// TIA Portal project "motors8" (V17)

(* hardware
DEVICE "S7-1500/ET200MP station_1"  S7-1500 station
   slot 0: "Rail_0"  Rack  6ES7 590-1***0-0AA0
   slot 1: "PLC_1"  CPU 1515-2 PN  6ES7 515-2AM02-0AB0  V2.9
      slot 3: "CPU display_1"  6ES7591-1BA00-0AA0
      slot 32768: "PROFINET interface_1"  X1
         slot 32769: "Port_1"  X1 P1
         slot 32770: "Port_2"  X1 P2
      slot 33024: "PROFINET interface_2"  X2
         slot 33025: "Port_1"  X2 P1
      slot 34817: "Virtual CP interface port_1"  Virtual CP interface port  Virtual CP interface port
   slot 2: "DQ 32x24VDC/0.5A BA_1"  DQ 32x24VDC/0.5A BA  6ES7 522-1BL10-0AA0  V1.1
DEVICE "PC-System_1"  SIMATIC PC station
   slot 0: "SIMATIC PC station"  Rail  SIMATIC PC-Station  V1.0
      slot 125: "Stationmanager"  Station_Manager  V6.0.4
   slot 1: "HMI_RT_1"  WinCC RT Advanced  6AV2 104-0xxxx-xxxx  17.0.0.0
      slot 33792: "Computer interface"  Host interface
   slot 2: "IE general_1"  IE General  IE_CP  V8.2.0
      slot 1: "PROFINET interface"  IEGeneral.Interface.8.2.0
*)

// ===== PLC "PLC_1"  CPU 1515-2 PN =====

VAR_GLOBAL   // PLC tag table "Default tag table"
   "MOTOR1" AT %Q0.0 : Bool;
   "MOTOR2" AT %Q0.1 : Bool;
   "MOTOR3" AT %Q0.2 : Bool;
   "MOTOR4" AT %Q0.3 : Bool;
   "MOTOR5" AT %Q0.4 : Bool;
   "MOTOR6" AT %Q0.5 : Bool;
   "MOTOR7" AT %Q0.6 : Bool;
   "MOTOR8" AT %Q0.7 : Bool;
END_VAR

TYPE "MotorLibrary"
   STRUCT
      "BREAKER ON" : Bool;
      OVERLOAD : Bool;
      CONTACTOR : Bool;
      "LED RUN" : Bool;
      "LED STOP" : Bool;
      "LED OVERLOAD" : Bool;
      "EMERGENCY STOP" : Bool;
      "START BUTTON" : Bool;
      "STOP BUTTON" : Bool;
      "RESET OVERLOAD" : Bool;
   END_STRUCT;
END_TYPE

DATA_BLOCK "MOTORsDB"   // DB1
{ S7_Optimized_Access := 'FALSE' }
VERSION : 0.1
   VAR
      M1 : "MotorLibrary";
      M2 : "MotorLibrary";
      M3 : "MotorLibrary";
      M4 : "MotorLibrary";
      M5 : "MotorLibrary";
      M6 : "MotorLibrary";
      M7 : "MotorLibrary";
      M8 : "MotorLibrary";
   END_VAR
BEGIN
END_DATA_BLOCK

DATA_BLOCK "FB_MOTOR1"   // DB2
{ S7_Optimized_Access := 'TRUE' }
VERSION : 0.1
// stored: InstanceOfName MOTORsLOGIC
"MOTORsLOGIC"
BEGIN
END_DATA_BLOCK

DATA_BLOCK "FB_MOTOR2"   // DB3
{ S7_Optimized_Access := 'TRUE' }
VERSION : 0.1
// stored: InstanceOfName MOTORsLOGIC
"MOTORsLOGIC"
BEGIN
END_DATA_BLOCK

DATA_BLOCK "FB_MOTOR3"   // DB4
{ S7_Optimized_Access := 'TRUE' }
VERSION : 0.1
// stored: InstanceOfName MOTORsLOGIC
"MOTORsLOGIC"
BEGIN
END_DATA_BLOCK

DATA_BLOCK "FB_MOTOR4"   // DB5
{ S7_Optimized_Access := 'TRUE' }
VERSION : 0.1
// stored: InstanceOfName MOTORsLOGIC
"MOTORsLOGIC"
BEGIN
END_DATA_BLOCK

DATA_BLOCK "FB_MOTOR5"   // DB6
{ S7_Optimized_Access := 'TRUE' }
VERSION : 0.1
// stored: InstanceOfName MOTORsLOGIC
"MOTORsLOGIC"
BEGIN
END_DATA_BLOCK

DATA_BLOCK "FB_MOTOR6"   // DB7
{ S7_Optimized_Access := 'TRUE' }
VERSION : 0.1
// stored: InstanceOfName MOTORsLOGIC
"MOTORsLOGIC"
BEGIN
END_DATA_BLOCK

DATA_BLOCK "FB_MOTOR7"   // DB8
{ S7_Optimized_Access := 'TRUE' }
VERSION : 0.1
// stored: InstanceOfName MOTORsLOGIC
"MOTORsLOGIC"
BEGIN
END_DATA_BLOCK

DATA_BLOCK "FB_MOTOR8"   // DB9
{ S7_Optimized_Access := 'TRUE' }
VERSION : 0.1
// stored: InstanceOfName MOTORsLOGIC
"MOTORsLOGIC"
BEGIN
END_DATA_BLOCK

FUNCTION_BLOCK "MOTORsLOGIC"   // FB1, LAD
{ S7_Optimized_Access := 'TRUE' }
VERSION : 0.1
   VAR_INPUT
      "BREAKER ON" : Bool;
      "EMERGENCY STOP" : Bool;
      "START BUTTON" : Bool;
      "STOP BUTTON" : Bool;
      "OVERLOAD RELAY" : Bool;
      "RESET OVERLOAD" : Bool;
   END_VAR
   VAR_OUTPUT
      CONTACTOR : Bool;
      "PLC OUTPUT" : Bool;
      "LED STOP" : Bool;
      "LED RUN" : Bool;
      "LED OVERLOAD" : Bool;
   END_VAR
   VAR_TEMP   // added for the SCL form of the ladder/FBD networks
      _w1 : Bool;
   END_VAR
BEGIN

REGION Network 1: Motors Logic Control
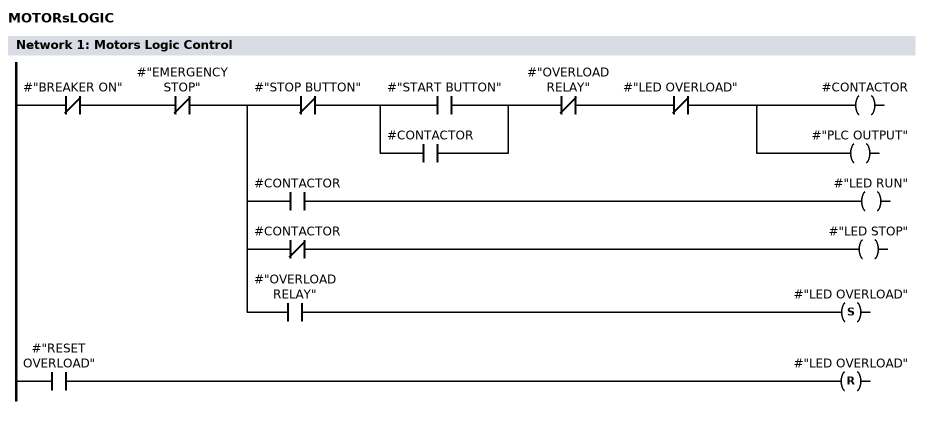
   RUNG wire#powerrail
      I_Contact( #"BREAKER ON" )
      I_Contact( #"EMERGENCY STOP" )
      wire#w1
      I_Contact( #"STOP BUTTON" )
      wire#w2
      Contact( #"START BUTTON" )
      wire#w3
      I_Contact( #"OVERLOAD RELAY" )
      I_Contact( #"LED OVERLOAD" )
      wire#w4
      Coil( #CONTACTOR )
   END_RUNG
   RUNG wire#w2
      Contact( #CONTACTOR )
   END_RUNG wire#w3
   RUNG wire#w4
      Coil( #"PLC OUTPUT" )
   END_RUNG
   RUNG wire#w1
      Contact( #CONTACTOR )
      Coil( #"LED RUN" )
   END_RUNG
   RUNG wire#w1
      I_Contact( #CONTACTOR )
      Coil( #"LED STOP" )
   END_RUNG
   RUNG wire#w1
      Contact( #"OVERLOAD RELAY" )
      S_Coil( #"LED OVERLOAD" )
   END_RUNG
   RUNG wire#powerrail
      Contact( #"RESET OVERLOAD" )
      R_Coil( #"LED OVERLOAD" )
   END_RUNG
   // the same network as SCL:
   #_w1 := NOT #"BREAKER ON" AND NOT #"EMERGENCY STOP";
   #CONTACTOR := #_w1 AND NOT #"STOP BUTTON" AND (#"START BUTTON" OR #CONTACTOR) AND NOT #"OVERLOAD RELAY" AND NOT #"LED OVERLOAD";
   #"PLC OUTPUT" := #CONTACTOR;
   #"LED RUN" := #_w1 AND #CONTACTOR;
   #"LED STOP" := #_w1 AND NOT #CONTACTOR;
   IF #_w1 AND #"OVERLOAD RELAY" THEN #"LED OVERLOAD" := TRUE; END_IF;
   IF #"RESET OVERLOAD" THEN #"LED OVERLOAD" := FALSE; END_IF;
END_REGION
END_FUNCTION_BLOCK

ORGANIZATION_BLOCK "Main"   // OB1, LAD, ProgramCycle
TITLE = "Main Program Sweep (Cycle)"
{ S7_Optimized_Access := 'TRUE' }
VERSION : 0.1
   VAR_INPUT
      Initial_Call : Bool;   // Initial call of this OB
      Remanence : Bool;   // =True, if remanent data are available
   END_VAR
BEGIN

REGION Network 1: MOTOR1
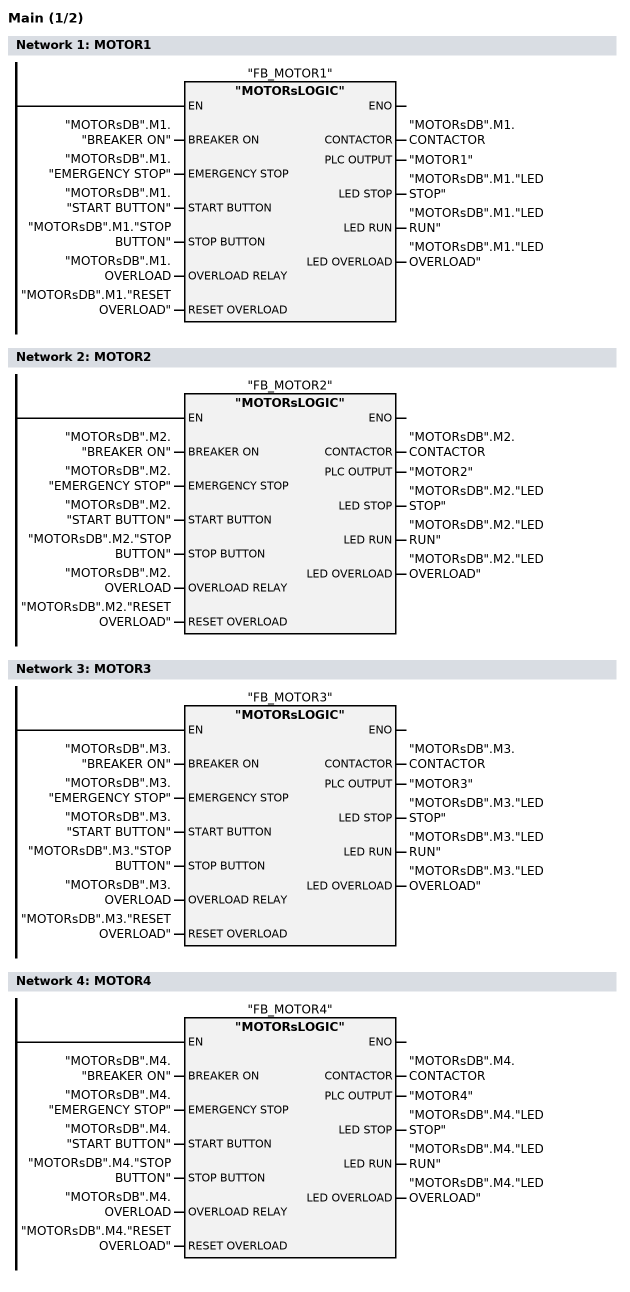
   RUNG wire#powerrail
      "FB_MOTOR1"("BREAKER ON" := "MOTORsDB".M1."BREAKER ON", "EMERGENCY STOP" := "MOTORsDB".M1."EMERGENCY STOP", "START BUTTON" := "MOTORsDB".M1."START BUTTON", "STOP BUTTON" := "MOTORsDB".M1."STOP BUTTON", "OVERLOAD RELAY" := "MOTORsDB".M1.OVERLOAD, "RESET OVERLOAD" := "MOTORsDB".M1."RESET OVERLOAD", CONTACTOR => "MOTORsDB".M1.CONTACTOR, "PLC OUTPUT" => "MOTOR1", "LED STOP" => "MOTORsDB".M1."LED STOP", "LED RUN" => "MOTORsDB".M1."LED RUN", "LED OVERLOAD" => "MOTORsDB".M1."LED OVERLOAD")
   END_RUNG
   // the same network as SCL:
   "FB_MOTOR1"("BREAKER ON" := "MOTORsDB".M1."BREAKER ON",   // "MOTORsLOGIC"
               "EMERGENCY STOP" := "MOTORsDB".M1."EMERGENCY STOP",
               "START BUTTON" := "MOTORsDB".M1."START BUTTON",
               "STOP BUTTON" := "MOTORsDB".M1."STOP BUTTON",
               "OVERLOAD RELAY" := "MOTORsDB".M1.OVERLOAD,
               "RESET OVERLOAD" := "MOTORsDB".M1."RESET OVERLOAD",
               CONTACTOR => "MOTORsDB".M1.CONTACTOR,
               "PLC OUTPUT" => "MOTOR1",
               "LED STOP" => "MOTORsDB".M1."LED STOP",
               "LED RUN" => "MOTORsDB".M1."LED RUN",
               "LED OVERLOAD" => "MOTORsDB".M1."LED OVERLOAD");
END_REGION

REGION Network 2: MOTOR2
   RUNG wire#powerrail
      "FB_MOTOR2"("BREAKER ON" := "MOTORsDB".M2."BREAKER ON", "EMERGENCY STOP" := "MOTORsDB".M2."EMERGENCY STOP", "START BUTTON" := "MOTORsDB".M2."START BUTTON", "STOP BUTTON" := "MOTORsDB".M2."STOP BUTTON", "OVERLOAD RELAY" := "MOTORsDB".M2.OVERLOAD, "RESET OVERLOAD" := "MOTORsDB".M2."RESET OVERLOAD", CONTACTOR => "MOTORsDB".M2.CONTACTOR, "PLC OUTPUT" => "MOTOR2", "LED STOP" => "MOTORsDB".M2."LED STOP", "LED RUN" => "MOTORsDB".M2."LED RUN", "LED OVERLOAD" => "MOTORsDB".M2."LED OVERLOAD")
   END_RUNG
   // the same network as SCL:
   "FB_MOTOR2"("BREAKER ON" := "MOTORsDB".M2."BREAKER ON",   // "MOTORsLOGIC"
               "EMERGENCY STOP" := "MOTORsDB".M2."EMERGENCY STOP",
               "START BUTTON" := "MOTORsDB".M2."START BUTTON",
               "STOP BUTTON" := "MOTORsDB".M2."STOP BUTTON",
               "OVERLOAD RELAY" := "MOTORsDB".M2.OVERLOAD,
               "RESET OVERLOAD" := "MOTORsDB".M2."RESET OVERLOAD",
               CONTACTOR => "MOTORsDB".M2.CONTACTOR,
               "PLC OUTPUT" => "MOTOR2",
               "LED STOP" => "MOTORsDB".M2."LED STOP",
               "LED RUN" => "MOTORsDB".M2."LED RUN",
               "LED OVERLOAD" => "MOTORsDB".M2."LED OVERLOAD");
END_REGION

REGION Network 3: MOTOR3
   RUNG wire#powerrail
      "FB_MOTOR3"("BREAKER ON" := "MOTORsDB".M3."BREAKER ON", "EMERGENCY STOP" := "MOTORsDB".M3."EMERGENCY STOP", "START BUTTON" := "MOTORsDB".M3."START BUTTON", "STOP BUTTON" := "MOTORsDB".M3."STOP BUTTON", "OVERLOAD RELAY" := "MOTORsDB".M3.OVERLOAD, "RESET OVERLOAD" := "MOTORsDB".M3."RESET OVERLOAD", CONTACTOR => "MOTORsDB".M3.CONTACTOR, "PLC OUTPUT" => "MOTOR3", "LED STOP" => "MOTORsDB".M3."LED STOP", "LED RUN" => "MOTORsDB".M3."LED RUN", "LED OVERLOAD" => "MOTORsDB".M3."LED OVERLOAD")
   END_RUNG
   // the same network as SCL:
   "FB_MOTOR3"("BREAKER ON" := "MOTORsDB".M3."BREAKER ON",   // "MOTORsLOGIC"
               "EMERGENCY STOP" := "MOTORsDB".M3."EMERGENCY STOP",
               "START BUTTON" := "MOTORsDB".M3."START BUTTON",
               "STOP BUTTON" := "MOTORsDB".M3."STOP BUTTON",
               "OVERLOAD RELAY" := "MOTORsDB".M3.OVERLOAD,
               "RESET OVERLOAD" := "MOTORsDB".M3."RESET OVERLOAD",
               CONTACTOR => "MOTORsDB".M3.CONTACTOR,
               "PLC OUTPUT" => "MOTOR3",
               "LED STOP" => "MOTORsDB".M3."LED STOP",
               "LED RUN" => "MOTORsDB".M3."LED RUN",
               "LED OVERLOAD" => "MOTORsDB".M3."LED OVERLOAD");
END_REGION

REGION Network 4: MOTOR4
   RUNG wire#powerrail
      "FB_MOTOR4"("BREAKER ON" := "MOTORsDB".M4."BREAKER ON", "EMERGENCY STOP" := "MOTORsDB".M4."EMERGENCY STOP", "START BUTTON" := "MOTORsDB".M4."START BUTTON", "STOP BUTTON" := "MOTORsDB".M4."STOP BUTTON", "OVERLOAD RELAY" := "MOTORsDB".M4.OVERLOAD, "RESET OVERLOAD" := "MOTORsDB".M4."RESET OVERLOAD", CONTACTOR => "MOTORsDB".M4.CONTACTOR, "PLC OUTPUT" => "MOTOR4", "LED STOP" => "MOTORsDB".M4."LED STOP", "LED RUN" => "MOTORsDB".M4."LED RUN", "LED OVERLOAD" => "MOTORsDB".M4."LED OVERLOAD")
   END_RUNG
   // the same network as SCL:
   "FB_MOTOR4"("BREAKER ON" := "MOTORsDB".M4."BREAKER ON",   // "MOTORsLOGIC"
               "EMERGENCY STOP" := "MOTORsDB".M4."EMERGENCY STOP",
               "START BUTTON" := "MOTORsDB".M4."START BUTTON",
               "STOP BUTTON" := "MOTORsDB".M4."STOP BUTTON",
               "OVERLOAD RELAY" := "MOTORsDB".M4.OVERLOAD,
               "RESET OVERLOAD" := "MOTORsDB".M4."RESET OVERLOAD",
               CONTACTOR => "MOTORsDB".M4.CONTACTOR,
               "PLC OUTPUT" => "MOTOR4",
               "LED STOP" => "MOTORsDB".M4."LED STOP",
               "LED RUN" => "MOTORsDB".M4."LED RUN",
               "LED OVERLOAD" => "MOTORsDB".M4."LED OVERLOAD");
END_REGION

REGION Network 5: MOTOR5
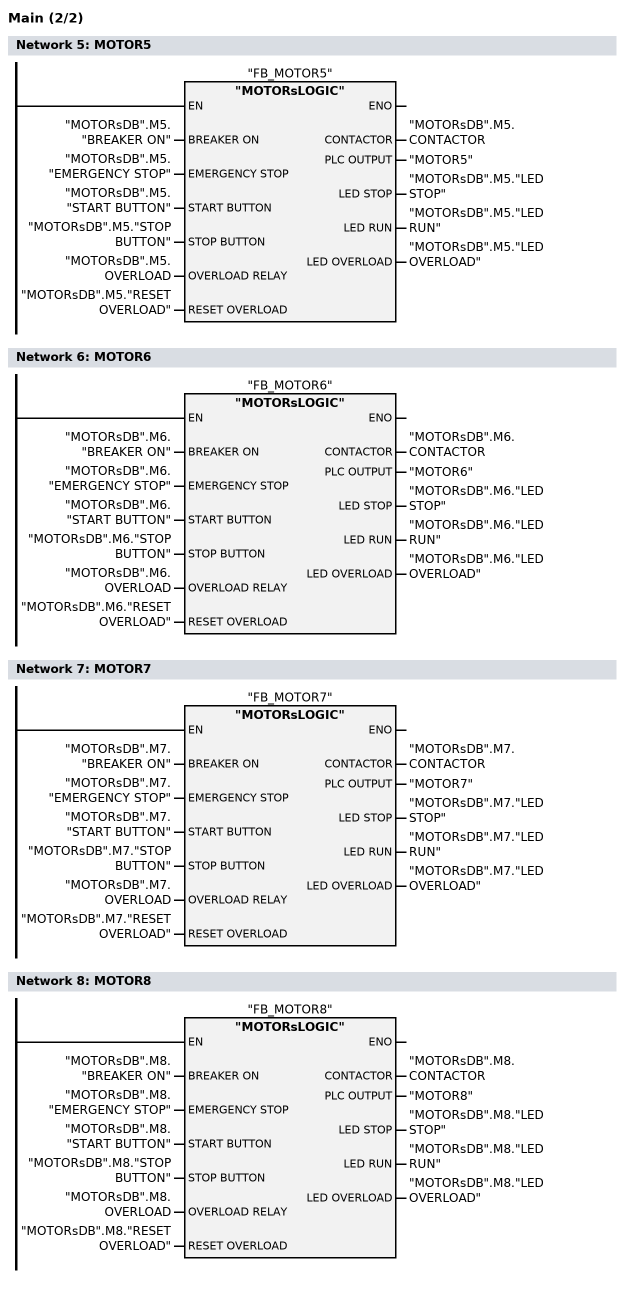
   RUNG wire#powerrail
      "FB_MOTOR5"("BREAKER ON" := "MOTORsDB".M5."BREAKER ON", "EMERGENCY STOP" := "MOTORsDB".M5."EMERGENCY STOP", "START BUTTON" := "MOTORsDB".M5."START BUTTON", "STOP BUTTON" := "MOTORsDB".M5."STOP BUTTON", "OVERLOAD RELAY" := "MOTORsDB".M5.OVERLOAD, "RESET OVERLOAD" := "MOTORsDB".M5."RESET OVERLOAD", CONTACTOR => "MOTORsDB".M5.CONTACTOR, "PLC OUTPUT" => "MOTOR5", "LED STOP" => "MOTORsDB".M5."LED STOP", "LED RUN" => "MOTORsDB".M5."LED RUN", "LED OVERLOAD" => "MOTORsDB".M5."LED OVERLOAD")
   END_RUNG
   // the same network as SCL:
   "FB_MOTOR5"("BREAKER ON" := "MOTORsDB".M5."BREAKER ON",   // "MOTORsLOGIC"
               "EMERGENCY STOP" := "MOTORsDB".M5."EMERGENCY STOP",
               "START BUTTON" := "MOTORsDB".M5."START BUTTON",
               "STOP BUTTON" := "MOTORsDB".M5."STOP BUTTON",
               "OVERLOAD RELAY" := "MOTORsDB".M5.OVERLOAD,
               "RESET OVERLOAD" := "MOTORsDB".M5."RESET OVERLOAD",
               CONTACTOR => "MOTORsDB".M5.CONTACTOR,
               "PLC OUTPUT" => "MOTOR5",
               "LED STOP" => "MOTORsDB".M5."LED STOP",
               "LED RUN" => "MOTORsDB".M5."LED RUN",
               "LED OVERLOAD" => "MOTORsDB".M5."LED OVERLOAD");
END_REGION

REGION Network 6: MOTOR6
   RUNG wire#powerrail
      "FB_MOTOR6"("BREAKER ON" := "MOTORsDB".M6."BREAKER ON", "EMERGENCY STOP" := "MOTORsDB".M6."EMERGENCY STOP", "START BUTTON" := "MOTORsDB".M6."START BUTTON", "STOP BUTTON" := "MOTORsDB".M6."STOP BUTTON", "OVERLOAD RELAY" := "MOTORsDB".M6.OVERLOAD, "RESET OVERLOAD" := "MOTORsDB".M6."RESET OVERLOAD", CONTACTOR => "MOTORsDB".M6.CONTACTOR, "PLC OUTPUT" => "MOTOR6", "LED STOP" => "MOTORsDB".M6."LED STOP", "LED RUN" => "MOTORsDB".M6."LED RUN", "LED OVERLOAD" => "MOTORsDB".M6."LED OVERLOAD")
   END_RUNG
   // the same network as SCL:
   "FB_MOTOR6"("BREAKER ON" := "MOTORsDB".M6."BREAKER ON",   // "MOTORsLOGIC"
               "EMERGENCY STOP" := "MOTORsDB".M6."EMERGENCY STOP",
               "START BUTTON" := "MOTORsDB".M6."START BUTTON",
               "STOP BUTTON" := "MOTORsDB".M6."STOP BUTTON",
               "OVERLOAD RELAY" := "MOTORsDB".M6.OVERLOAD,
               "RESET OVERLOAD" := "MOTORsDB".M6."RESET OVERLOAD",
               CONTACTOR => "MOTORsDB".M6.CONTACTOR,
               "PLC OUTPUT" => "MOTOR6",
               "LED STOP" => "MOTORsDB".M6."LED STOP",
               "LED RUN" => "MOTORsDB".M6."LED RUN",
               "LED OVERLOAD" => "MOTORsDB".M6."LED OVERLOAD");
END_REGION

REGION Network 7: MOTOR7
   RUNG wire#powerrail
      "FB_MOTOR7"("BREAKER ON" := "MOTORsDB".M7."BREAKER ON", "EMERGENCY STOP" := "MOTORsDB".M7."EMERGENCY STOP", "START BUTTON" := "MOTORsDB".M7."START BUTTON", "STOP BUTTON" := "MOTORsDB".M7."STOP BUTTON", "OVERLOAD RELAY" := "MOTORsDB".M7.OVERLOAD, "RESET OVERLOAD" := "MOTORsDB".M7."RESET OVERLOAD", CONTACTOR => "MOTORsDB".M7.CONTACTOR, "PLC OUTPUT" => "MOTOR7", "LED STOP" => "MOTORsDB".M7."LED STOP", "LED RUN" => "MOTORsDB".M7."LED RUN", "LED OVERLOAD" => "MOTORsDB".M7."LED OVERLOAD")
   END_RUNG
   // the same network as SCL:
   "FB_MOTOR7"("BREAKER ON" := "MOTORsDB".M7."BREAKER ON",   // "MOTORsLOGIC"
               "EMERGENCY STOP" := "MOTORsDB".M7."EMERGENCY STOP",
               "START BUTTON" := "MOTORsDB".M7."START BUTTON",
               "STOP BUTTON" := "MOTORsDB".M7."STOP BUTTON",
               "OVERLOAD RELAY" := "MOTORsDB".M7.OVERLOAD,
               "RESET OVERLOAD" := "MOTORsDB".M7."RESET OVERLOAD",
               CONTACTOR => "MOTORsDB".M7.CONTACTOR,
               "PLC OUTPUT" => "MOTOR7",
               "LED STOP" => "MOTORsDB".M7."LED STOP",
               "LED RUN" => "MOTORsDB".M7."LED RUN",
               "LED OVERLOAD" => "MOTORsDB".M7."LED OVERLOAD");
END_REGION

REGION Network 8: MOTOR8
   RUNG wire#powerrail
      "FB_MOTOR8"("BREAKER ON" := "MOTORsDB".M8."BREAKER ON", "EMERGENCY STOP" := "MOTORsDB".M8."EMERGENCY STOP", "START BUTTON" := "MOTORsDB".M8."START BUTTON", "STOP BUTTON" := "MOTORsDB".M8."STOP BUTTON", "OVERLOAD RELAY" := "MOTORsDB".M8.OVERLOAD, "RESET OVERLOAD" := "MOTORsDB".M8."RESET OVERLOAD", CONTACTOR => "MOTORsDB".M8.CONTACTOR, "PLC OUTPUT" => "MOTOR8", "LED STOP" => "MOTORsDB".M8."LED STOP", "LED RUN" => "MOTORsDB".M8."LED RUN", "LED OVERLOAD" => "MOTORsDB".M8."LED OVERLOAD")
   END_RUNG
   // the same network as SCL:
   "FB_MOTOR8"("BREAKER ON" := "MOTORsDB".M8."BREAKER ON",   // "MOTORsLOGIC"
               "EMERGENCY STOP" := "MOTORsDB".M8."EMERGENCY STOP",
               "START BUTTON" := "MOTORsDB".M8."START BUTTON",
               "STOP BUTTON" := "MOTORsDB".M8."STOP BUTTON",
               "OVERLOAD RELAY" := "MOTORsDB".M8.OVERLOAD,
               "RESET OVERLOAD" := "MOTORsDB".M8."RESET OVERLOAD",
               CONTACTOR => "MOTORsDB".M8.CONTACTOR,
               "PLC OUTPUT" => "MOTOR8",
               "LED STOP" => "MOTORsDB".M8."LED STOP",
               "LED RUN" => "MOTORsDB".M8."LED RUN",
               "LED OVERLOAD" => "MOTORsDB".M8."LED OVERLOAD");
END_REGION
END_ORGANIZATION_BLOCK

(* ===== HMI "HMI_RT_1" =====
system functions are stored by id; their names below are inferred from use
connection "HMI_Connection_1": ETHERNET, S7_1500_OMS

HMI tags "Default tag table"
   "MOTORsDB_M1" : MotorLibrary = PLC MOTORsDB.M1 AT %DB1.DBX0.0, 1 s
   "MOTORsDB_M2" : MotorLibrary = PLC MOTORsDB.M2 AT %DB1.DBX2.0, 1 s
   "MOTORsDB_M3" : MotorLibrary = PLC MOTORsDB.M3 AT %DB1.DBX4.0, 1 s
   "MOTORsDB_M4" : MotorLibrary = PLC MOTORsDB.M4 AT %DB1.DBX6.0, 1 s
   "MOTORsDB_M5" : MotorLibrary = PLC MOTORsDB.M5 AT %DB1.DBX8.0, 1 s
   "MOTORsDB_M6" : MotorLibrary = PLC MOTORsDB.M6 AT %DB1.DBX10.0, 1 s
   "MOTORsDB_M7" : MotorLibrary = PLC MOTORsDB.M7 AT %DB1.DBX12.0, 1 s
   "MOTORsDB_M8" : MotorLibrary = PLC MOTORsDB.M8 AT %DB1.DBX14.0, 1 s

screen "MOTOR1 SCREEN" 1024x768
   ScreenModuleView "FACEPLATE1_1" at 63,34 size 908x595; ScreenModuleType ""; Guid_{11997190-6804} 'MOTOR1'
      Guid_{11997190-4317} <- "MOTORsDB_M1"
   Button "Button_1" at 37,657 size 116x67; TextOff 'MOTOR2'
      on Click: ActivateScreen("MOTOR2 SCREEN", 0)
   Button "Button_2" at 176,657 size 116x67; TextOff 'MOTOR3'
      on Click: ActivateScreen("MOTOR3 SCREEN", 0)
   Button "Button_3" at 315,657 size 116x67; TextOff 'MOTOR4'
      on Click: ActivateScreen("MOTOR4 SCREEN", 0)
   Button "Button_4" at 454,657 size 116x67; TextOff 'MOTOR5'
      on Click: ActivateScreen("MOTOR5 SCREEN", 0)
   Button "Button_5" at 593,657 size 116x67; TextOff 'MOTOR6'
      on Click: ActivateScreen("MOTOR6 SCREEN", 0)
   Button "Button_6" at 732,657 size 116x67; TextOff 'MOTOR7'
      on Click: ActivateScreen("MOTOR7 SCREEN", 0)
   Button "Button_7" at 871,657 size 116x67; TextOff 'MOTOR8'
      on Click: ActivateScreen("MOTOR8 SCREEN", 0)

screen "MOTOR2 SCREEN" 1024x768
   ScreenModuleView "FACEPLATE1_1" at 70,33 size 908x595; Guid_{11997190-6804} 'MOTOR2'; ScreenModuleType ""
      Guid_{11997190-4317} <- "MOTORsDB_M2"
   Button "Button_1" at 37,657 size 116x67; TextOff 'MOTOR1'
      on Click: ActivateScreen("MOTOR1 SCREEN", 0)
   Button "Button_2" at 176,657 size 116x67; TextOff 'MOTOR3'
      on Click: ActivateScreen("MOTOR3 SCREEN", 0)
   Button "Button_3" at 315,657 size 116x67; TextOff 'MOTOR4'
      on Click: ActivateScreen("MOTOR4 SCREEN", 0)
   Button "Button_4" at 454,657 size 116x67; TextOff 'MOTOR5'
      on Click: ActivateScreen("MOTOR5 SCREEN", 0)
   Button "Button_5" at 593,657 size 116x67; TextOff 'MOTOR6'
      on Click: ActivateScreen("MOTOR6 SCREEN", 0)
   Button "Button_6" at 732,657 size 116x67; TextOff 'MOTOR7'
      on Click: ActivateScreen("MOTOR7 SCREEN", 0)
   Button "Button_7" at 871,657 size 116x67; TextOff 'MOTOR8'
      on Click: ActivateScreen("MOTOR8 SCREEN", 0)

screen "MOTOR3 SCREEN" 1024x768
   ScreenModuleView "FACEPLATE1_1" at 63,34 size 908x595; Guid_{11997190-6804} 'MOTOR3'; ScreenModuleType ""
      Guid_{11997190-4317} <- "MOTORsDB_M3"
   Button "Button_1" at 37,657 size 116x67; TextOff 'MOTOR1'
      on Click: ActivateScreen("MOTOR1 SCREEN", 0)
   Button "Button_2" at 176,657 size 116x67; TextOff 'MOTOR2'
      on Click: ActivateScreen("MOTOR2 SCREEN", 0)
   Button "Button_3" at 315,657 size 116x67; TextOff 'MOTOR4'
      on Click: ActivateScreen("MOTOR4 SCREEN", 0)
   Button "Button_4" at 454,657 size 116x67; TextOff 'MOTOR5'
      on Click: ActivateScreen("MOTOR5 SCREEN", 0)
   Button "Button_5" at 593,657 size 116x67; TextOff 'MOTOR6'
      on Click: ActivateScreen("MOTOR6 SCREEN", 0)
   Button "Button_6" at 732,657 size 116x67; TextOff 'MOTOR7'
      on Click: ActivateScreen("MOTOR7 SCREEN", 0)
   Button "Button_7" at 871,657 size 116x67; TextOff 'MOTOR8'
      on Click: ActivateScreen("MOTOR8 SCREEN", 0)

screen "MOTOR4 SCREEN" 1024x768
   ScreenModuleView "FACEPLATE1_1" at 63,34 size 908x595; Guid_{11997190-6804} 'MOTOR4'; ScreenModuleType ""
      Guid_{11997190-4317} <- "MOTORsDB_M4"
   Button "Button_1" at 37,657 size 116x67; TextOff 'MOTOR1'
      on Click: ActivateScreen("MOTOR1 SCREEN", 0)
   Button "Button_2" at 176,657 size 116x67; TextOff 'MOTOR2'
      on Click: ActivateScreen("MOTOR2 SCREEN", 0)
   Button "Button_3" at 315,657 size 116x67; TextOff 'MOTOR3'
      on Click: ActivateScreen("MOTOR3 SCREEN", 0)
   Button "Button_4" at 454,657 size 116x67; TextOff 'MOTOR5'
      on Click: ActivateScreen("MOTOR5 SCREEN", 0)
   Button "Button_5" at 593,657 size 116x67; TextOff 'MOTOR6'
      on Click: ActivateScreen("MOTOR6 SCREEN", 0)
   Button "Button_6" at 732,657 size 116x67; TextOff 'MOTOR7'
      on Click: ActivateScreen("MOTOR7 SCREEN", 0)
   Button "Button_7" at 871,657 size 116x67; TextOff 'MOTOR8'
      on Click: ActivateScreen("MOTOR8 SCREEN", 0)

screen "MOTOR5 SCREEN" 1024x768
   ScreenModuleView "FACEPLATE1_1" at 63,34 size 908x595; Guid_{11997190-6804} 'MOTOR5'; ScreenModuleType ""
      Guid_{11997190-4317} <- "MOTORsDB_M5"
   Button "Button_1" at 37,657 size 116x67; TextOff 'MOTOR1'
      on Click: ActivateScreen("MOTOR1 SCREEN", 0)
   Button "Button_2" at 176,657 size 116x67; TextOff 'MOTOR2'
      on Click: ActivateScreen("MOTOR2 SCREEN", 0)
   Button "Button_3" at 315,657 size 116x67; TextOff 'MOTOR3'
      on Click: ActivateScreen("MOTOR3 SCREEN", 0)
   Button "Button_4" at 454,657 size 116x67; TextOff 'MOTOR4'
      on Click: ActivateScreen("MOTOR4 SCREEN", 0)
   Button "Button_5" at 593,657 size 116x67; TextOff 'MOTOR6'
      on Click: ActivateScreen("MOTOR6 SCREEN", 0)
   Button "Button_6" at 732,657 size 116x67; TextOff 'MOTOR7'
      on Click: ActivateScreen("MOTOR7 SCREEN", 0)
   Button "Button_7" at 871,657 size 116x67; TextOff 'MOTOR8'
      on Click: ActivateScreen("MOTOR8 SCREEN", 0)

screen "MOTOR6 SCREEN" 1024x768
   ScreenModuleView "FACEPLATE1_1" at 63,34 size 908x595; Guid_{11997190-6804} 'MOTOR6'; ScreenModuleType ""
      Guid_{11997190-4317} <- "MOTORsDB_M6"
   Button "Button_1" at 37,657 size 116x67; TextOff 'MOTOR1'
      on Click: ActivateScreen("MOTOR1 SCREEN", 0)
   Button "Button_2" at 176,657 size 116x67; TextOff 'MOTOR2'
      on Click: ActivateScreen("MOTOR2 SCREEN", 0)
   Button "Button_3" at 315,657 size 116x67; TextOff 'MOTOR3'
      on Click: ActivateScreen("MOTOR3 SCREEN", 0)
   Button "Button_4" at 454,657 size 116x67; TextOff 'MOTOR4'
      on Click: ActivateScreen("MOTOR4 SCREEN", 0)
   Button "Button_5" at 593,657 size 116x67; TextOff 'MOTOR5'
      on Click: ActivateScreen("MOTOR5 SCREEN", 0)
   Button "Button_6" at 732,657 size 116x67; TextOff 'MOTOR7'
      on Click: ActivateScreen("MOTOR7 SCREEN", 0)
   Button "Button_7" at 871,657 size 116x67; TextOff 'MOTOR8'
      on Click: ActivateScreen("MOTOR8 SCREEN", 0)

screen "MOTOR7 SCREEN" 1024x768
   ScreenModuleView "FACEPLATE1_1" at 63,34 size 908x595; Guid_{11997190-6804} 'MOTOR7'; ScreenModuleType ""
      Guid_{11997190-4317} <- "MOTORsDB_M7"
   Button "Button_1" at 37,657 size 116x67; TextOff 'MOTOR1'
      on Click: ActivateScreen("MOTOR1 SCREEN", 0)
   Button "Button_2" at 176,657 size 116x67; TextOff 'MOTOR2'
      on Click: ActivateScreen("MOTOR2 SCREEN", 0)
   Button "Button_3" at 315,657 size 116x67; TextOff 'MOTOR3'
      on Click: ActivateScreen("MOTOR3 SCREEN", 0)
   Button "Button_4" at 454,657 size 116x67; TextOff 'MOTOR4'
      on Click: ActivateScreen("MOTOR4 SCREEN", 0)
   Button "Button_5" at 593,657 size 116x67; TextOff 'MOTOR5'
      on Click: ActivateScreen("MOTOR5 SCREEN", 0)
   Button "Button_6" at 732,657 size 116x67; TextOff 'MOTOR6'
      on Click: ActivateScreen("MOTOR6 SCREEN", 0)
   Button "Button_7" at 871,657 size 116x67; TextOff 'MOTOR8'
      on Click: ActivateScreen("MOTOR8 SCREEN", 0)

screen "MOTOR8 SCREEN" 1024x768
   ScreenModuleView "FACEPLATE1_1" at 63,34 size 908x595; Guid_{11997190-6804} 'MOTOR8'; ScreenModuleType ""
      Guid_{11997190-4317} <- "MOTORsDB_M8"
   Button "Button_1" at 37,657 size 116x67; TextOff 'MOTOR1'
      on Click: ActivateScreen("MOTOR1 SCREEN", 0)
   Button "Button_2" at 176,657 size 116x67; TextOff 'MOTOR2'
      on Click: ActivateScreen("MOTOR2 SCREEN", 0)
   Button "Button_3" at 315,657 size 116x67; TextOff 'MOTOR3'
      on Click: ActivateScreen("MOTOR3 SCREEN", 0)
   Button "Button_4" at 454,657 size 116x67; TextOff 'MOTOR4'
      on Click: ActivateScreen("MOTOR4 SCREEN", 0)
   Button "Button_5" at 593,657 size 116x67; TextOff 'MOTOR5'
      on Click: ActivateScreen("MOTOR5 SCREEN", 0)
   Button "Button_6" at 732,657 size 116x67; TextOff 'MOTOR6'
      on Click: ActivateScreen("MOTOR6 SCREEN", 0)
   Button "Button_7" at 871,657 size 116x67; TextOff 'MOTOR7'
      on Click: ActivateScreen("MOTOR7 SCREEN", 0)
*)

(* ===== HMI "HMI_RT_1" =====
system functions are stored by id; their names below are inferred from use

ScreenModuleEditorView "FACEPLATE1" 1050x800
   Switch "Switch_1" at 53,182 size 75x56; TextOn 'ON'; CaptionText 'TURN CB'; TextOff 'OFF'
      on SwitchOff: ResetBit("MLIB.BREAKER ON")
      on SwitchOn: SetBit("MLIB.BREAKER ON")
   Switch "Switch_2" at 55,429 size 80x60; TextOn 'ON'; CaptionText 'TEST OL'; TextOff 'OFF'
      on SwitchOff: ResetBit("MLIB.OVERLOAD")
      on SwitchOn: SetBit("MLIB.OVERLOAD")
   SymbolLibrary "Symbol library_1" at 143,527 size 225x105
      Appearance <- "MLIB.LED RUN"
   Button "Button_1" at 346,258 size 48x35; TextOff 'FU1'
   Button "Button_2" at 506,258 size 48x35; TextOff 'FU2'
   TextField "Text field_1" at 701,184 size 27x22; Text 'EM'
   TextField "Text field_2" at 700,280 size 25x22; Text 'B1'
   TextField "Text field_3" at 678,446 size 26x22; Text 'OL'
   TextField "Text field_4" at 680,361 size 25x22; Text 'B2'
   TextField "Text field_5" at 771,364 size 28x22; Text 'KM'
   Button "Button_3" at 631,550 size 74x49; TextOff 'KM'
      Appearance <- "MLIB.CONTACTOR"
   Circle "Circle_3" at 789,117 size 48x48
      Appearance <- "MLIB.LED STOP"
   Circle "Circle_4" at 861,115 size 48x48
      Appearance <- "MLIB.LED RUN"
   Circle "Circle_5" at 932,115 size 48x48
      Appearance <- "MLIB.LED OVERLOAD"
   Button "Button_4" at 787,174 size 96x51; TextOff 'START'
      on Press: function_b14e0dd5("MLIB.START BUTTON", 0)
   Button "Button_5" at 894,174 size 96x52; TextOff 'STOP'
      on Press: function_b14e0dd5("MLIB.STOP BUTTON", 0)
   Button "Button_6" at 789,228 size 96x51; TextOff 'EM-STOP'
      on Press: function_b14e0dd5("MLIB.EMERGENCY STOP", 0)
   Button "Button_7" at 896,228 size 96x51; TextOff 'RST'
      on Press: function_b14e0dd5("MLIB.RESET OVERLOAD", 0)
   TextField "Text field_8" at 789,95 size 46x22; Text 'STOP'
   TextField "Text field_9" at 861,95 size 39x22; Text 'RUN'
   TextField "Text field_10" at 939,94 size 26x22; Text 'OL'
   TextField "Text field_11" at 432,243 size 35x22; Text 'TR1'
   TextField "Text field_12" at 329,320 size 134x22; Text '380VAC/220VAC'
   TextField "Text field_13" at 778,64 size 205x22; Text 'MOTOR1 CONTROL PANEL'
   TextField "Text field_6" at 389,17 size 24x22; Text 'L1'
   TextField "Text field_7" at 389,39 size 24x22; Text 'L2'
   TextField "Text field_14" at 389,63 size 24x22; Text 'L3'
   TextField "Text field_15" at 389,91 size 16x22; Text 'G'
   TextField "Text field_16" at 53,43 size 65x22; Text '380VAC'
   TextField "Text field_17" at 168,633 size 62x22; Text 'MOTOR'
   TextField "Text field_18" at 99,344 size 28x22; Text 'KM'
   Line "Line_11" at 151,193 size 28x55
      Visibility <- "MLIB.BREAKER ON"
   Line "Line_12" at 207,189 size 25x53
      Visibility <- "MLIB.BREAKER ON"
   Line "Line_13" at 262,191 size 30x56
      Visibility <- "MLIB.BREAKER ON"
   Line "Line_17" at 150,343 size 28x55
      Visibility <- "MLIB.LED RUN"
   Line "Line_18" at 206,339 size 25x53
      Visibility <- "MLIB.LED RUN"
   Line "Line_19" at 261,341 size 30x56
      Visibility <- "MLIB.LED RUN"
   Line "Line_22" at 177,340 size 1x52
      Visibility <- "MLIB.LED RUN"
   Line "Line_23" at 239,337 size 1x52
      Visibility <- "MLIB.LED RUN"
   Line "Line_24" at 295,337 size 1x52
      Visibility <- "MLIB.LED RUN"
   Line "Line_25" at 292,188 size 1x52
      Visibility <- "MLIB.BREAKER ON"
   Line "Line_26" at 230,187 size 1x52
      Visibility <- "MLIB.BREAKER ON"
   Line "Line_27" at 178,190 size 1x52
      Visibility <- "MLIB.BREAKER ON"
   Line "Line_49" at 663,187 size 15x31
      Visibility <- "MLIB.EMERGENCY STOP"
   Line "Line_52" at 662,283 size 15x31
      Visibility <- "MLIB.STOP BUTTON"
   Line "Line_56" at 666,471 size 30x1
      Visibility <- "MLIB.OVERLOAD"
   Line "Line_65" at 646,361 size 19x29
      Visibility <- "MLIB.START BUTTON"
   Line "Line_78" at 663,350 size 2x40
      Visibility <- "MLIB.START BUTTON"
*)

(* ===== HMI "HMI_RT_1" =====
system functions are stored by id; their names below are inferred from use

ScreenModuleEditorView "FACEPLATE1" 1050x800
   Switch "Switch_1" at 53,182 size 75x56; TextOn 'ON'; CaptionText 'TURN CB'; TextOff 'OFF'
      on SwitchOn: SetBit("MLIB.BREAKER ON")
      on SwitchOff: ResetBit("MLIB.BREAKER ON")
   Switch "Switch_2" at 55,429 size 80x60; TextOn 'ON'; CaptionText 'TEST OL'; TextOff 'OFF'
      on SwitchOn: SetBit("MLIB.OVERLOAD")
      on SwitchOff: ResetBit("MLIB.OVERLOAD")
   SymbolLibrary "Symbol library_1" at 143,527 size 225x105
      Appearance <- "MLIB.LED RUN"
   Button "Button_1" at 346,258 size 48x35; TextOff 'FU1'
   Button "Button_2" at 506,258 size 48x35; TextOff 'FU2'
   TextField "Text field_1" at 701,184 size 27x22; Text 'EM'
   TextField "Text field_2" at 700,280 size 25x22; Text 'B1'
   TextField "Text field_3" at 678,446 size 26x22; Text 'OL'
   TextField "Text field_4" at 680,361 size 25x22; Text 'B2'
   TextField "Text field_5" at 771,364 size 28x22; Text 'KM'
   Button "Button_3" at 631,550 size 74x49; TextOff 'KM'
      Appearance <- "MLIB.CONTACTOR"
   Circle "Circle_3" at 789,117 size 48x48
      Appearance <- "MLIB.LED STOP"
   Circle "Circle_4" at 861,115 size 48x48
      Appearance <- "MLIB.LED RUN"
   Circle "Circle_5" at 932,115 size 48x48
      Appearance <- "MLIB.LED OVERLOAD"
   Button "Button_4" at 787,174 size 96x51; TextOff 'START'
      on Press: function_b14e0dd5("MLIB.START BUTTON", 0)
   Button "Button_5" at 894,174 size 96x52; TextOff 'STOP'
      on Press: function_b14e0dd5("MLIB.STOP BUTTON", 0)
   Button "Button_6" at 789,228 size 96x51; TextOff 'EM-STOP'
      on Press: function_b14e0dd5("MLIB.EMERGENCY STOP", 0)
   Button "Button_7" at 896,228 size 96x51; TextOff 'RST'
      on Press: function_b14e0dd5("MLIB.RESET OVERLOAD", 0)
   TextField "Text field_8" at 789,95 size 46x22; Text 'STOP'
   TextField "Text field_9" at 861,95 size 39x22; Text 'RUN'
   TextField "Text field_10" at 939,94 size 26x22; Text 'OL'
   TextField "Text field_11" at 432,243 size 35x22; Text 'TR1'
   TextField "Text field_12" at 329,320 size 134x22; Text '380VAC/220VAC'
   TextField "Text field_13" at 778,64 size 205x22; Text 'MOTOR1 CONTROL PANEL'
   TextField "Text field_6" at 389,17 size 24x22; Text 'L1'
   TextField "Text field_7" at 389,39 size 24x22; Text 'L2'
   TextField "Text field_14" at 389,63 size 24x22; Text 'L3'
   TextField "Text field_15" at 389,91 size 16x22; Text 'G'
   TextField "Text field_16" at 53,43 size 65x22; Text '380VAC'
   TextField "Text field_17" at 168,633 size 62x22; Text 'MOTOR'
   TextField "Text field_18" at 99,344 size 28x22; Text 'KM'
   TextField "Text field_19" at 350,671 size 100x34; Text 'MNAME'
   Line "Line_11" at 151,193 size 28x55
      Visibility <- "MLIB.BREAKER ON"
   Line "Line_12" at 207,189 size 25x53
      Visibility <- "MLIB.BREAKER ON"
   Line "Line_13" at 262,191 size 30x56
      Visibility <- "MLIB.BREAKER ON"
   Line "Line_17" at 150,343 size 28x55
      Visibility <- "MLIB.LED RUN"
   Line "Line_18" at 206,339 size 25x53
      Visibility <- "MLIB.LED RUN"
   Line "Line_19" at 261,341 size 30x56
      Visibility <- "MLIB.LED RUN"
   Line "Line_22" at 177,340 size 1x52
      Visibility <- "MLIB.LED RUN"
   Line "Line_23" at 239,337 size 1x52
      Visibility <- "MLIB.LED RUN"
   Line "Line_24" at 295,337 size 1x52
      Visibility <- "MLIB.LED RUN"
   Line "Line_25" at 292,188 size 1x52
      Visibility <- "MLIB.BREAKER ON"
   Line "Line_26" at 230,187 size 1x52
      Visibility <- "MLIB.BREAKER ON"
   Line "Line_27" at 178,190 size 1x52
      Visibility <- "MLIB.BREAKER ON"
   Line "Line_49" at 663,187 size 15x31
      Visibility <- "MLIB.EMERGENCY STOP"
   Line "Line_52" at 662,283 size 15x31
      Visibility <- "MLIB.STOP BUTTON"
   Line "Line_56" at 666,471 size 30x1
      Visibility <- "MLIB.OVERLOAD"
   Line "Line_65" at 646,361 size 19x29
      Visibility <- "MLIB.START BUTTON"
   Line "Line_78" at 663,350 size 2x40
      Visibility <- "MLIB.START BUTTON"
*)